(* CODESYS project EmiconEventsControl.library
   Author: Emicon
   Placeholder: EmiconEvtCtl
   Title: Emicon Events Control
   Version: 3.5.17.20
   DefaultNamespace: EMEvtCtl
   Company: Emicon

Project tree, tasks and I/O mapping:
  libraries: CmpEventMgr, * (System); Standard, * (System); SysTypes Interfaces, * (System); CmpApp, 3.5.17.0 (System)
  global variables EventIDs
*)

// EventIDs
VAR_GLOBAL CONSTANT
	CMPID_EM_EVT_CTL		: DWORD := 16#163F2010;
	EVT_B_BUTTON_PRESSED 	: DWORD := 16#10001;
	EVT_GPIO_50 			: DWORD := 16#10002;
	EVT_GPIO_51 			: DWORD := 16#10003;
	EVT_GPIO_52 			: DWORD := 16#10004;
	EVT_GPIO_53 			: DWORD := 16#10005;
END_VAR
